// TIA Portal V19 export
DATA_BLOCK "CallEquipment_DB"   // DB14
AUTHOR : Siemens_FA_SUP
// stored: InstanceOfName Unit2.EM2.CallEquipment, InstanceOfType FB, Namespace Unit2.EM2
"Unit2.EM2.CallEquipment"
   // VAR_IN_OUT
   //    unitStatus : "LAF_typeUnitStatus";
   //    unitAlarmDB : "LAF_typeAlarms";
   //    emFeedback : "LUC_typeEmFeedback";
   // END_VAR
   // VAR
   //    statUnitStatus { ExternalWritable := 'False'} : "LAF_typeUnitStatus";
   //    instJobExecute { ExternalWritable := 'False'} : "LAF_SelectJob";
   //    instJobStopping { ExternalWritable := 'False'; S7_SetPoint := 'True'} : "LAF_SelectJob";
   //    instJobStarting { ExternalWritable := 'False'; S7_SetPoint := 'True'} : "LAF_SelectJob";
   //    instJobHolding { ExternalWritable := 'False'; S7_SetPoint := 'True'} : "LAF_SelectJob";
   //    instJobUnHolding { ExternalWritable := 'False'; S7_SetPoint := 'True'} : "LAF_SelectJob";
   //    instJobReseting { ExternalWritable := 'False'; S7_SetPoint := 'True'} : "LAF_SelectJob";
   //    instSequence { ExternalWritable := 'False'} : "Unit2.EM2.Sequence";
   //    instManageBitAlarms { ExternalWritable := 'False'} : "LAF_ManageBitAlarms";
   //    instCmReset { ExternalWritable := 'False'; S7_SetPoint := 'True'} : "Unit2.EM2.EXCHANGETRAY_ConstraintRollerCmResetOperator";
   //    instcm1Vfd206 { ExternalWritable := 'False'} : "LEXCHANGETRAY_RollerVfd";
   //    instcm6SignalTM { ExternalWritable := 'False'; S7_SetPoint := 'True'} : "LEXCHANGETRAY_U2Em2SingleTM";
   //    instCm5AxisPos { ExternalWritable := 'False'} : "LBC_AxisSimpleControl";
   //    instCm2TrayLiftingCylinder { ExternalWritable := 'False'; S7_SetPoint := 'True'} : "LEXCHANGETRAY_Cylinder";
   //    instCm3CellLiftingCylinder { ExternalWritable := 'False'; S7_SetPoint := 'True'} : "LEXCHANGETRAY_Cylinder";
   //    instCm4PositioningPinCylinder { ExternalWritable := 'False'; S7_SetPoint := 'True'} : "LEXCHANGETRAY_Cylinder";
   //    instCm7Pc { ExternalWritable := 'False'; S7_SetPoint := 'True'} : "LEXCHANGETRAY_PcAcuator";
   //    instCm8Scanner { ExternalWritable := 'False'} : "LEXCHANGETRAY_Sr1000_Profinet";
   //    statLstUnitMode { ExternalWritable := 'False'; S7_SetPoint := 'True'} : DInt;
   // END_VAR
BEGIN
END_DATA_BLOCK
